// TIA Portal V19 export
FUNCTION "DATE& TIME" : Void   // FC8, LAD
{ S7_Optimized_Access := 'TRUE' }
// stored: SetENOAutomatically false
BEGIN

REGION Network 1
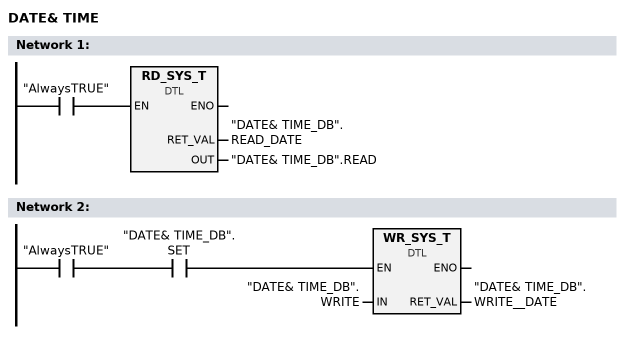
   RUNG wire#powerrail
      Contact( "AlwaysTRUE" )
      { S7_Templates := "date_type := DTL" } RD_SYS_T(RET_VAL => "DATE& TIME_DB".READ_DATE, OUT => "DATE& TIME_DB".READ)
   END_RUNG
   // the same network as SCL:
   IF "AlwaysTRUE" THEN "DATE& TIME_DB".READ_DATE := RD_SYS_T(OUT => "DATE& TIME_DB".READ); END_IF;
END_REGION

REGION Network 2
   RUNG wire#powerrail
      Contact( "AlwaysTRUE" )
      Contact( "DATE& TIME_DB".SET )
      { S7_Templates := "date_type := DTL" } WR_SYS_T(IN := "DATE& TIME_DB".WRITE, RET_VAL => "DATE& TIME_DB".WRITE__DATE)
   END_RUNG
   // the same network as SCL:
   IF "AlwaysTRUE" AND "DATE& TIME_DB".SET THEN
       "DATE& TIME_DB".WRITE__DATE := WR_SYS_T(IN := "DATE& TIME_DB".WRITE);
   END_IF;
END_REGION
END_FUNCTION
